FUNCTION_BLOCK "FB_ClockGen"
{ S7_Optimized_Access := 'TRUE' }
VERSION : 0.1

// FB_ClockGen: gera dois bits de pisca (ondas quadradas ~50% duty) para sinalizacao
// (consumidos pelo FB_MachineMode: torre amarela/vermelha, luz de Reset).
// REQUER chamada incondicional TODO scan (ex.: OB1): o auto-rearme do TON e o toggle de
// estado dependem disso — nao mover para OB de evento sem revisar. Periodo real =
// 2x meio-periodo (+ ~2 scans, desprezivel). Dominio esperado: Hz > 0 e moderado
// (ex.: 0,5-10 Hz); Hz <= 0 -> saida FALSE; Hz muito alto degrada o clock (sem teto aqui).
    VAR_INPUT
        i_SlowHz : LReal;   // frequência do pisca lento (Hz) — ex. Cfg.ClkSlowHz = 1.0
        i_FastHz : LReal;   // frequência do pisca rápido (Hz) — ex. Cfg.ClkFastHz = 3.0
    END_VAR

    VAR_OUTPUT
        o_Slow : Bool;      // onda quadrada lenta (~1 Hz)
        o_Fast : Bool;      // onda quadrada rápida (~3 Hz)
    END_VAR

    VAR
        s_tSlow : TON_TIME;   // temporizador do meio-período lento
        s_tFast : TON_TIME;   // temporizador do meio-período rápido
        s_SlowState : Bool := TRUE;   // nível atual da onda lenta (alternado); parte em TRUE p/ acender no 1o scan
        s_FastState : Bool := TRUE;   // nível atual da onda rápida (alternado); idem — blinda "torre apagada na partida"
    END_VAR

    VAR_TEMP
        t_halfSlow : LReal;       // meio-período lento em ms
        t_halfFast : LReal;       // meio-período rápido em ms
    END_VAR

BEGIN

    REGION Pisca lento
    // Gera onda quadrada ~50% duty a partir de i_SlowHz
        // meio-período (ms) = 1000 / (2 * Hz); período total = 1/Hz.
        // FALLBACK fail-safe: Hz <= 0 (config ausente/zerada) NAO apaga a sinalizacao —
        // usa 1 Hz padrao. Perder o pisca da torre por config 0 e anti-fail-safe (a
        // emergencia/falha ficaria sem indicacao visivel). Evita tambem divisao por zero.
        IF #i_SlowHz > 0.0 THEN
            #t_halfSlow := 1000.0 / (2.0 * #i_SlowHz);
        ELSE
            #t_halfSlow := 500.0;   // 1 Hz (meio-periodo 500 ms)
        END_IF;
        // TON auto-rearmado: Q pulsa 1 scan a cada meio-período
        #s_tSlow(IN := NOT #s_tSlow.Q,
        PT := DINT_TO_TIME(LREAL_TO_DINT(#t_halfSlow)));
        // a cada pulso de Q, inverte o nível -> onda quadrada
        IF #s_tSlow.Q THEN
            #s_SlowState := NOT #s_SlowState;
        END_IF;
        #o_Slow := #s_SlowState;
    END_REGION

    REGION Pisca rapido
    // Gera onda quadrada ~50% duty a partir de i_FastHz
        // meio-período (ms) = 1000 / (2 * Hz); período total = 1/Hz.
        // FALLBACK fail-safe: Hz <= 0 -> usa 3 Hz padrao (ver justificativa no pisca lento).
        IF #i_FastHz > 0.0 THEN
            #t_halfFast := 1000.0 / (2.0 * #i_FastHz);
        ELSE
            #t_halfFast := 166.0;   // ~3 Hz (meio-periodo ~166 ms)
        END_IF;
        // TON auto-rearmado: Q pulsa 1 scan a cada meio-período
        #s_tFast(IN := NOT #s_tFast.Q,
        PT := DINT_TO_TIME(LREAL_TO_DINT(#t_halfFast)));
        // a cada pulso de Q, inverte o nível -> onda quadrada
        IF #s_tFast.Q THEN
            #s_FastState := NOT #s_FastState;
        END_IF;
        #o_Fast := #s_FastState;
    END_REGION

END_FUNCTION_BLOCK
